TYPE CoverPanelProcesses :
STRUCT
	///Start opening the panel
	startOpening: Process;
	///Start closing the panel
	startClosing: Process;
END_STRUCT
END_TYPE

(* stored: Version 1.1.0.1, ProductVersion 3.1.4019.2
   DUT CoverPanelProcesses: Id {e0c26258-fc78-4203-8aac-352236bde119} *)
